FUNCTION_BLOCK Xts EXTENDS PML_Method_Base
VAR
	_homePosition : MC_LREAL;
	_HomeSpeed : MC_LREAL;
	mcCollisionGroup : CollisionGroup;
	_XtsTrackHardware : IXtsHardware;
	XtsHwState : XtsHardwareState;
	EnableSequence : XtsEnableSequence(mcCollisionGroup);
	DisableSequence : XtsDisableSequence(mcCollisionGroup);
	State : UINT;	
	i : UINT;
	AtHome: BOOL;
	_tracks : UINT;
	_MoverArray : ARRAY[1..SystemParameters.NumberOfMovers] OF IMover;
END_VAR

{analysis -2}

METHOD PROTECTED Aborting : BOOL
VAR
	
END_VAR
CASE State OF
	0:
		DisableSequence.Disable();
		State := 1;
			
	1:
		IF DisableSequence.Done THEN
			State := 0;
			ipackml.SetStateComplete();
			Aborting := TRUE;
		END_IF
	ELSE
		Aborting := FALSE;
END_CASE
END_METHOD

METHOD PUBLIC ActivateTracksInMovers : BOOL
VAR
	TmsMoverInterface : ITmsMover;
	ActivateTrackResult : BOOL;
END_VAR
FOR i := 1 TO SystemParameters.NumberOfMovers DO
	IF __QUERYINTERFACE(_MoverArray[i],TmsMoverInterface) THEN
		ActivateTrackResult := TmsMoverInterface.ActivateTrack(newTrack := TmsMoverInterface.ActiveTrack);
	END_IF
END_FOR
ActivateTracksInMovers := true;
END_METHOD

METHOD PROTECTED Clearing : BOOL
VAR_INPUT
END_VAR
CASE State OF
	0:
		IF EnableSequence.Enable() THEN
			State := 1;
		END_IF	
		
	1:
		IF EnableSequence.Done THEN
			State := 2;
		END_IF
		
	2:
		IF ActivateTracksInMovers() THEN
			ipackml.SetStateComplete();
			State := 0;
			Clearing := TRUE;
		END_IF
	ELSE
		Clearing := FALSE;
END_CASE
END_METHOD

METHOD PUBLIC Cycle : HRESULT
VAR
	EnableResult : HRESULT;
	DisableResult : HRESULT;
	GrpStopResult : HRESULT;
	CollisionResult : HRESULT;
END_VAR
Cycle := SUPER^.Cycle();
EnableResult := EnableSequence.Cycle();
DisableResult := DisableSequence.Cycle();
GrpStopResult := GroupStop.Cycle();
CollisionResult := mcCollisionGroup.Cycle();

IF EnableResult = E_FAIL OR
	DisableResult = E_FAIL OR
	GrpStopResult = E_FAIL OR
	CollisionResult = E_FAIL THEN
	Cycle := E_FAIL;
END_IF
END_METHOD

METHOD FB_init : BOOL
VAR_INPUT
	bInitRetains : BOOL; // if TRUE, the retain variables are initialized (warm start / cold start)
	bInCopyCode : BOOL;  // if TRUE, the instance afterwards gets moved into the copy code (online change)
	XtsRunner : I_XtsRunner;
END_VAR
XtsRunner.AddComponent(THIS^);
END_METHOD

METHOD PUBLIC GetTMSMoverInterface : BOOL
VAR_INPUT
END_VAR
VAR
	TmsMoverInterface : ITmsMover;
END_VAR
FOR i := 1 TO SystemParameters.NumberOfMovers DO
	IF __QUERYINTERFACE(_MoverArray[i],TmsMoverInterface) THEN
		TmsMoverInterface.SetMoverInterface(MoverInterface := _XtsTrackHardware.GetMoverEnvInterface(i));
	END_IF
END_FOR
END_METHOD

PROPERTY PUBLIC HomePosition : mc_lreal
GET
HomePosition := _homePosition;
END_GET
SET
_homePosition := HomePosition;
END_SET
END_PROPERTY

PROPERTY HomeSpeed : mc_lreal
GET
HomeSpeed := _HomeSpeed;
END_GET
SET
_HomeSpeed := HomeSpeed;
END_SET
END_PROPERTY

PROPERTY MoverArray : array[1..SystemParameters.NumberOfMovers] of IMover
GET
MoverArray := _MoverArray;
END_GET
SET
_MoverArray := MoverArray;
EnableSequence.MoverArray := MoverArray;
DisableSequence.MoverArray := MoverArray;
END_SET
END_PROPERTY

METHOD PUBLIC MoverHomeSequence : BOOL
VAR_INPUT
END_VAR
FOR i := 1 TO SystemParameters.NumberOfMovers DO
	_MoverArray[i].MoveTo(Position := _homePosition, Velocity := _HomeSpeed, BackwardMove := FALSE);
END_FOR 
MoverHomeSequence := TRUE;
END_METHOD

METHOD PROTECTED Resetting : BOOL
VAR_INPUT
END_VAR
CASE State OF
	0:
		IF MoverHomeSequence() THEN
			State := 1;
		END_IF
	
	1:
		AtHome := TRUE;
		FOR i := 1 TO SystemParameters.NumberOfMovers DO
				AtHome := AtHome AND _MoverArray[i].isStationary();
		END_FOR 
		IF AtHome THEN
			State := 0;
			ipackml.SetStateComplete();	
			Resetting := TRUE;
		END_IF
	ELSE
		Resetting := FALSE;	
END_CASE
END_METHOD

METHOD PROTECTED Stopping : BOOL
VAR_INPUT
END_VAR
CASE State OF
	0:
		mcCollisionGroup.GroupStop();
		State := 1;
		
	1:
		IF mcCollisionGroup.GroupState = CAGroupStatus.mcGroupStateStandby THEN
			State := 0;
			ipackml.SetStateComplete();
			Stopping := TRUE;
		END_IF
	ELSE
		Stopping := FALSE;
END_CASE
END_METHOD

PROPERTY PUBLIC Tracks : UINT
GET
Tracks := _tracks;
END_GET
SET
_tracks := Tracks;
END_SET
END_PROPERTY

METHOD PROTECTED Undefined : BOOL
VAR_INPUT
END_VAR
CASE XtsHwState OF
	XtsHardwareState.Init:
		IF _XtsTrackHardware.SetTracksForDetection() THEN
			XtsHwState := XtsHardwareState.Redetect;
		END_IF
		
	XtsHardwareState.Redetect:
		IF _XtsTrackHardware.TriggerMoverDetection() THEN
			XtsHwState := XtsHardwareState.MoversValid;
		END_IF
		
	XtsHardwareState.MoversValid:
		IF _XtsTrackHardware.getAllMoversValid() THEN
			XtsHwState := XtsHardwareState.AllMoversFound;
		END_IF
	
	XtsHardwareState.AllMoversFound:
		IF _XtsTrackHardware.getMoversDetected() THEN
			XtsHwState := XtsHardwareState.XTSMode;
		END_IF
		
	XtsHardwareState.XTSMode:
		IF _XtsTrackHardware.IsInSim() THEN
			XtsHwState := XtsHardwareState.MoverIdDetection;
		ELSE
			XtsHwState := XtsHardwareState.CheckModuleVoltages;
		END_IF
		
	XtsHardwareState.CheckModuleVoltages:
		IF _XtsTrackHardware.Is24VdcOK() = 2 AND _XtsTrackHardware.Is48VdcOK() = 2 THEN
			XtsHwState := XtsHardwareState.MoverIdDetection;
		END_IF
	
	XtsHardwareState.MoverIdDetection:
		IF _XtsTrackHardware.TriggerMoverID() THEN
			XtsHwState := XtsHardwareState.HWReady;
			GetTMSMoverInterface();
			ipackml.PmlStateCommand(Command := E_PMLCommand.ePMLCommand_Abort);
		END_IF
	
	XtsHardwareState.HWReady:
		
		
END_CASE
END_METHOD

PROPERTY XtsTrackHardware : IXtsHardware
GET
XtsTrackHardware := _XtsTrackHardware;
END_GET
SET
_XtsTrackHardware := XtsTrackHardware;
END_SET
END_PROPERTY

END_FUNCTION_BLOCK

(* stored: Version 1.1.0.1, ProductVersion 3.1.4024.12
   POU Xts: Id {4538c683-94fc-49a1-b5ad-30ffec5e4eff}, SpecialFunc None
   Folder Action States: Id {52cebbbe-42d9-490e-86b9-bf5151fd8965}
   Folder Operations: Id {0e8598c4-3d58-4c14-a12f-6fd3f3ea02bf}
   Folder Wait States: Id {63f323b6-e159-475d-b0ee-857bfb772605}
   Method Aborting: Id {f4025447-c7fa-4c21-bcd4-655228f2af38}
   Method ActivateTracksInMovers: Id {682f2d4e-bf73-44bf-93e3-716a6d45755c}
   Method Clearing: Id {7ebb7a7d-7271-4f69-b79f-9ca8eeb5c574}
   Method Cycle: Id {da42838e-fb00-40a5-96f4-b787aa883566}
   Method FB_init: Id {7656e6f5-212b-4fe7-8cf3-636ae6db9244}
   Method GetTMSMoverInterface: Id {0e64eced-3444-47ea-9660-c818e7a9dea9}
   Property HomePosition: Id {7488af26-181d-46aa-9621-c1c9bb1f6cd2}
   Get Get: Id {204400f9-e0e2-4b38-927a-449ec513969c}
   Set Set: Id {21b02a35-3878-4951-a8db-c2a9a5cebc6f}
   Property HomeSpeed: Id {1d1b8038-88e9-4101-981d-99bed1ba5b18}
   Get Get: Id {0a3ad8ef-2031-4e74-8b6e-8a654900fd7a}
   Set Set: Id {ddb9be5e-d4fd-4d3d-a099-37476a9afab3}
   Property MoverArray: Id {5c1cfa9c-be49-4324-bcf5-1be968bfce44}
   Get Get: Id {2b512b99-b3b1-44cb-bf62-7cd45f8e95a6}
   Set Set: Id {806f65c3-00a8-4311-b6e2-aa6af5313c87}
   Method MoverHomeSequence: Id {5c2deb91-ebd0-4a93-99ec-6a6bbbd5e076}
   Method Resetting: Id {284a2a86-6aa9-45b7-b9c4-39c067c7a709}
   Method Stopping: Id {3cd6a931-8a7e-487a-9f0d-8a2db098be82}
   Property Tracks: Id {8eb8f4ad-907d-4ff8-9789-8832cf169bda}
   Get Get: Id {92aead6c-a657-4c6b-8c96-d2980dde0d91}
   Set Set: Id {a91cec47-6d8c-44af-ab33-578bdff8cace}
   Method Undefined: Id {a91364b7-9260-4707-a829-905210de4834}
   Property XtsTrackHardware: Id {10aeacae-a746-485a-b0e8-a2e9fb26c42b}
   Get Get: Id {b51a74ba-fecc-49a6-94a3-853ee17e2470}
   Set Set: Id {2e7570c1-50ca-40b9-8c5b-c0e86681ca7a} *)
